// TIA Portal V20 export
VAR_GLOBAL   // PLC tag table "Default tag table"
   Start AT %I0.0 : Bool;
   Stop AT %I0.1 : Bool;
   Process_on AT %Q0.0 : Bool;
   AutoON AT %M100.0 : Bool;   // AutoON
   Complete_Program_1 AT %Q100.1 : Bool;
END_VAR
